(* CoDeSys 2.3 export: E_TEMPERATUREUNIT.EXP *)

(* Data type *)
TYPE E_TemperatureUnit : (
	KELVIN,
	GRAD_CELSIUS,
	GRAD_FAHRENHEIT,
	GRAD_RANKINE,
	GRAD_DELISLE,
	GRAD_REAUMUR,
	GRAD_NEWTON,
	GRAD_ROMER
);
END_TYPE
